FUNCTION TryConvert_LWORD_TO_WORD : BOOL
VAR_INPUT
	in : LWORD;
	out : REFERENCE TO WORD;
END_VAR

IF in > DatatypeLimits.MAX_VALUE_OF_LWORD_WHICH_CAN_BE_HELD_IN_A_WORD THEN
	RETURN;
END_IF

out := LWORD_TO_WORD(in);
TryConvert_LWORD_TO_WORD := TRUE;

END_FUNCTION

(* stored: Version 1.1.0.1, ProductVersion 3.1.4024.12
   POU TryConvert_LWORD_TO_WORD: Id {ccf40431-fb9e-45c7-9379-2389678c19c1}, SpecialFunc None *)
